// TIA Portal V20 export
DATA_BLOCK "LAF_InternalManual"   // DB43
VERSION : 19.0
// stored: MemoryReserve 100
   VAR
      hmi : Array[1..1] of "LAF_typeManHmiDisp";   // Anzahl der HMIs - modifizieren Sie die Array-Größe auf Basis der erforderlichen HMI / number of HMIs - modify the array size based on the required HMIs / número de HMI: modificar el tamaño del array según las HMI requeridas / nombre d'IHM - modifier la taille du tableau en fonction du nombre d'IHM requis / numero di HMI - modificare la dimensione di array in base alle HMI richieste / HMI 수 - 필요한 HMI에 따라 배열 크기를 수정합니다. / HMI 数量 - 根据所需的 HMI 修改数组大小
      manualOperationEnabled : Bool;   // feedback whether the manual operation lines are selected
      emsWithManualOpConfigured { ExternalWritable := 'False'} : "LGM_emsWithManualOpConfigured";   // List of EMs with manual operation configured, for HMI button visibility
      disableUnit1 { S7_SetPoint := 'True'} : Bool;
      RisingEdge : Bool;
   END_VAR
BEGIN
END_DATA_BLOCK
